FUNCTION_BLOCK BLIND_SCENE
VAR_INPUT
	UP, DN : BOOL;
	S_IN : BYTE;
	PI, AI : BYTE;
	ENABLE : BOOL;
	SWRITE : BOOL;
	SCENE : BYTE;
END_VAR
VAR_OUTPUT
	QU, QD : BOOL;
	STATUS : BYTE;
	PO, AO : BYTE;
END_VAR
VAR RETAIN
	sx : ARRAY[0..15,0..2] OF BYTE;
END_VAR
VAR_TEMP
	x : BYTE;
END_VAR

(*
version 1.1	29. jan 2008
programmer 	hugo
tested by		tobias


*)

(* delete all bits except the lower 4 of scene *)
x := scene AND 16#0F;

IF enable AND sx[x,2] > 0 AND UP AND DN THEN
	po := sx[x,0];
	ao := sx[x,1];
	status := 160 + x;  (* Status number is 160 to 175 for the 16 scenes *)
	QU := TRUE;
	QD := TRUE;
ELSE
	QU := UP;
	QD := DN;
	status := S_IN;
	po := pi;
	ao := ai;
END_IF;

(* write scene if necessary *)
IF swrite THEN
	status := 176;		(* write scene *)
	sx[x,0] := pi;
	sx[x,1] := ai;
	IF enable THEN sx[x,2] := 1; ELSE sx[x,2] := 0; END_IF; (* if sx[x,2] = 0 the scene is disabled *)
END_IF;


(* revision history
hm	24. oct 2007	rev 1.0
	original release

hm		29.1.2008	rev 1.1
	replaced shr/shl with and for better performance
*)

END_FUNCTION_BLOCK

(* stored: Version 1.1.0.1, ProductVersion 3.1.4024.9
   POU BLIND_SCENE: Id {20c74de8-79a1-4461-91ca-ffc53e0c55a3}, SpecialFunc None *)
